PROGRAM myCNC_Call_BogieIndex
VAR
END_VAR

END_PROGRAM

(* stored: Version 1.1.0.1, ProductVersion 3.1.4024.11
   POU myCNC_Call_BogieIndex: Id {d5095a9d-5bbc-4bff-9db1-1835808bbb83}, SpecialFunc None *)
